// TIA Portal V20 export
DATA_BLOCK "EmNodes"   // DB146
// Global DB for the data exchange between the module levels (Between Unit and EM or EM and CM)
// stored: Access Published, MemoryReserve 100, Namespace Unit1
   VAR
      unitStatus { ExternalWritable := 'False'} : "LAF_typeUnitStatus";   // Status of the unit
      emFeedback { ExternalWritable := 'False'} : Array[0.._.U1_NO_OF_EMs] of "LUC_typeEmFeedback";   // Status of the individual equipment modules
      emRelations { ExternalWritable := 'False'} : Struct
         em00 { S7_SetPoint := 'True'} : "Unit1.type_emRelations_em0";
         em01 { S7_SetPoint := 'True'} : "Unit1.type_emRelations_em1";
         em02 { S7_SetPoint := 'True'} : "Unit1.type_emRelations_em2";
         em03 { S7_SetPoint := 'True'} : "Unit1.type_emRelations_em3";
         em04 { S7_SetPoint := 'True'} : "Unit1.type_emRelations_em4";
         em05 { S7_SetPoint := 'True'} : "Unit1.type_emRelations_em5";
         em06 { S7_SetPoint := 'True'} : "Unit1.type_emRelations_em6";
         em07 { S7_SetPoint := 'True'} : "Unit1.type_emRelations_em7";
         em08 { S7_SetPoint := 'True'} : "Unit1.type_emRelations_em8";
         em09 { S7_SetPoint := 'True'} : "Unit1.type_emRelations_em9";
         em10 { S7_SetPoint := 'True'} : "Unit1.type_emRelations_em10";
         em11 { S7_SetPoint := 'True'} : "Unit1.type_emRelations_em11";
         em12 { S7_SetPoint := 'True'} : "Unit1.type_emRelations_em12";
         em13 { S7_SetPoint := 'True'} : "Unit1.type_emRelations_em13";
      END_STRUCT;
      emIt1 : Array[0..13] of "LER_OEM_Data";
      emIt2 : Array[0..13] of "LER_OEM_Data";
      enableControlInterfaces { ExternalWritable := 'False'} : "LAF_typeEnableControlInterfaces";
      oem { S7_SetPoint := 'True'} : Array[0..10] of "LER_OEM_Data";
      FATModeSelect { ExternalWritable := 'False'} : "LER_TypeFATMode_ModeSelect";
      FATModeInterface { ExternalWritable := 'False'} : "LER_TypeFATModeInterface";
      signalStack { ExternalWritable := 'False'} : "LUC_typeSignalStackByBool";
      clock { ExternalWritable := 'False'} : "LAF_typeGlobalClockMem";
      sleep : Struct
         State { S7_SetPoint := 'True'} : "LER_typeSleepMode";
         command { S7_SetPoint := 'True'} : "LER_typeSleep";
      END_STRUCT;
      DryRunDataStatusCheck : Array[0..7] of Bool;
      SpecialFunctionMode : Struct
         EM0_JRdetectPV : Array[0..15] of Bool;
         EM1_JRdetectPV : Array[0..15] of Bool;
         EM2_JRdetectPV : Array[0..15] of Bool;
         EM3_JRdetectPV : Array[0..15] of Bool;
         EM4_JRdetectPV : Array[0..15] of Bool;
         EM5_JRdetectPV : Array[0..15] of Bool;
         EM6_JRdetectPV : Array[0..15] of Bool;
         EM7_JRdetectPV : Array[0..15] of Bool;
         EM8_JRdetectPV : Array[0..15] of Bool;
         EM9_JRdetectPV : Array[0..15] of Bool;
         EM10_JRdetectPV : Array[0..15] of Bool;
         EM11_JRdetectPV : Array[0..15] of Bool;
         EM12_JRdetectPV : Array[0..15] of Bool;
         EM13_JRdetectPV : Array[0..15] of Bool;
      END_STRUCT;
      motionOFF : Struct
         DR1 : Bool;
         DR2 : Bool;
         DR3 : Bool;
         DR4 : Bool;
         DR5 : Bool;
         DR6 : Bool;
         DR7 : Bool;
         DR8 : Bool;
         DR9 : Bool;
         DR10 : Bool;
         DR11 : Bool;
         DR12 : Bool;
         DR13 : Bool;
         DR14 : Bool;
         DR15 : Bool;
         DR16 : Bool;
         DR17 : Bool;
         DR18 : Bool;
         DR19 : Bool;
         DR20 : Bool;
      END_STRUCT;
      slmRunning { ExternalWritable := 'False'} : Bool;
      slmPowerOff { ExternalWritable := 'False'} : Bool;
      InterfaceTestMode { ExternalWritable := 'False'} : Bool;
      CapabilityModeComplete { ExternalWritable := 'False'} : Bool;
      SamplingModeComplete { ExternalWritable := 'False'} : Bool;
      stateCommandsExecute { ExternalWritable := 'False'} : Bool;
      unitAnyDoorUnlock { ExternalWritable := 'False'} : Bool;
      emAnyDoorUnlock : Bool;
      SleepModeActivationTime : Time;
      DeepSleepModeActivationTime : Time;
      SleepModeChangeReq : Bool;
      DeepSleepModeChangeReq : Bool;
      WakeupRecoveryRequired : Bool;
      "========Communication========" { ExternalWritable := 'False'} : Bool;
      BA010 : "LER_typeCommunication";
      BA015 : "LER_typeCommunication";
      BA030 : "LER_typeCommunication";
      BA040 : "LER_typeCommunication";
      BA100 { S7_SetPoint := 'True'} : "LER_type_mzc_Communication";
      UnitCommunication : Struct
         ToConveyorA : "LER_typeCommunicationData_Conveyor";
         FromConveyorA : "LER_typeCommunicationData_Conveyor";
      END_STRUCT;
      "========Safety========" { ExternalWritable := 'False'} : Bool;
      devicesSummary : "LWONIK_typeDevicesStatusSummary";
      safetyZone1OpEnable { ExternalWritable := 'False'} : "LWONIK_typeSafetyZoneManualOperation";
      safetyStatusZone1 : "LWONIK_typeZoneStatus";
      mainOpMode { ExternalWritable := 'False'} : "LWONIK_typeOperationMode";
      pHmiMode { ExternalWritable := 'False'} : "LWONIK_typePhmiMode";
      ScsMode { ExternalWritable := 'False'} : "LWONIK_typeScsMode";
      ScrapBox1 : "LWONIK_typeScrapBox";
      ScrapBox2 : "LWONIK_typeScrapBox";
      ScrapBox3 : "LWONIK_typeScrapBox";
      FdoorStatus { ExternalWritable := 'False'} : "LWONIK_typeFromSafetyDoorStatus";
      EstopStatus { ExternalWritable := 'False'} : "LWONIK_typeFromSafetyEstopStatus";
      OPLampStatus : "LWONIK_typeToSafetyLampStatus";
      doorOpenRequest { ExternalWritable := 'False'} : Bool;
      "=======ETC========" : Bool;
      unitRecipe { ExternalWritable := 'False'} : "LER_typeUnitRecipe";
      unitInterface { ExternalWritable := 'False'} : Struct
         stack1AndNgBox1 { S7_SetPoint := 'True'} : "LER_typeBeforeInterface";
         Stack1AndOutPP : "LER_typeBeforeInterface";
         stack2AndNgBox2 { S7_SetPoint := 'True'} : "LER_typeBeforeInterface";
         Stack2AndOutPP { S7_SetPoint := 'True'} : "LER_typeBeforeInterface";
      END_STRUCT;
      emDistance { ExternalWritable := 'False'} : Array[1..2] of "LER_typeDistanceInterface";
      allBrakeTest { ExternalWritable := 'False'} : "LER_typeBrakeTestUnitInterface";
      temperature { ExternalWritable := 'False'} : Struct
         hotPressLeft : Struct
            doorOpenOK : "Safety.typeHotPressTempOk";
         END_STRUCT;
         hotPressRight : Struct
            doorOpenOK : "Safety.typeHotPressTempOk";
         END_STRUCT;
      END_STRUCT;
      MQTT : "LMQTT_typeDB";
      powerMeter { S7_SetPoint := 'True'} : "LSicar_typeEnMeterVisuStruct";
      MobilePanelConnected : Bool;
      "=====Only Engineer Used=====" { ExternalAccessible := 'False'; ExternalVisible := 'False'; ExternalWritable := 'False'} : Bool;
      historyDataAllClear { ExternalAccessible := 'False'; ExternalVisible := 'False'; ExternalWritable := 'False'} : Bool;
      simulationMode { ExternalWritable := 'False'} : Bool;
   END_VAR
BEGIN
   emRelations.em03.LReal."01" := 1000000.0;
   emRelations.em04.LReal."01" := 1000000.0;
   // DryRunDataStatusCheck[0] : True : Part OK / false : Part NG
   // DryRunDataStatusCheck[2] : True : always NG
   // DryRunDataStatusCheck[3] : True : always OK
   BA030.StackToInspection.UnitStatus.state.stopped := TRUE;
   BA030.StackToInspection.InterfaceData."Bool"[4] := TRUE;
   BA030.StackToInspection.InterfaceData."Bool"[51] := TRUE;
   BA040.StackToInspection.UnitStatus.state.stopped := TRUE;
   BA040.StackToInspection.InterfaceData."Bool"[4] := TRUE;
   BA040.StackToInspection.InterfaceData."Bool"[51] := TRUE;
   // UnitCommunication.ToConveyorA.InterfaceData."Bool"[0] : Heartbeat
   // UnitCommunication.ToConveyorA.InterfaceData."Bool"[1] : ReadyForOperation
   // UnitCommunication.ToConveyorA.InterfaceData."Bool"[2] : MachineInOperation
   // UnitCommunication.ToConveyorA.InterfaceData."Bool"[3] : NoInterference
   // UnitCommunication.ToConveyorA.InterfaceData."Bool"[10] : PartOn
   // UnitCommunication.ToConveyorA.InterfaceData."Bool"[11] : PartReady
   // UnitCommunication.ToConveyorA.InterfaceData."Bool"[20] : LoaderOutsideModule
   // UnitCommunication.ToConveyorA.InterfaceData."Bool"[21] : LoaderOutsideCollision
   // UnitCommunication.ToConveyorA.InterfaceData."Bool"[22] : RequestCollisionON
   // UnitCommunication.ToConveyorA.InterfaceData."Bool"[30] : UnloadRun
   // UnitCommunication.ToConveyorA.InterfaceData."Bool"[31] : QrReadReady
   // UnitCommunication.ToConveyorA.InterfaceData."Bool"[32] : UnloadReady
   // UnitCommunication.ToConveyorA.InterfaceData."Bool"[33] : UnloadComplete
   // UnitCommunication.FromConveyorA.InterfaceData."Bool"[0] : Heartbeat
   // UnitCommunication.FromConveyorA.InterfaceData."Bool"[1] : ReadyForOperation
   // UnitCommunication.FromConveyorA.InterfaceData."Bool"[2] : MachineInOperation
   // UnitCommunication.FromConveyorA.InterfaceData."Bool"[3] : NoInterference
   // UnitCommunication.FromConveyorA.InterfaceData."Bool"[10] : PartOn
   // UnitCommunication.FromConveyorA.InterfaceData."Bool"[11] : PartReady
   // UnitCommunication.FromConveyorA.InterfaceData."Bool"[20] : CollisionAreaOn
   // UnitCommunication.FromConveyorA.InterfaceData."Bool"[21] : CollisionAreaOff
   // UnitCommunication.FromConveyorA.InterfaceData."Bool"[30] : RequestPart
   // UnitCommunication.FromConveyorA.InterfaceData."Bool"[31] : QrReadComplete
   // UnitCommunication.FromConveyorA.InterfaceData."Bool"[32] : UngripRequest
   // UnitCommunication.FromConveyorA.InterfaceData."Bool"[33] : LoadComplete
   unitRecipe.unitRecipe.sideTaping1stCount := 2;
   unitRecipe.unitRecipe.sideTaping2ndCount := 1;
   unitRecipe.unitRecipe.sideTaping3rdCount := 1;
   unitRecipe.unitRecipe.sideTaping4thCount := 1;
   // emDistance[1] : JR PP left ↔ right X-axis
   // emDistance[2] : Tranfer PP left ↔ right X-axis
   MQTT.connParam.broker := '192.168.1.246';
   MQTT.connParam.keepAlive := 60;
END_DATA_BLOCK
